// TIA Portal V17 export
// export: Created 2023-09-10T16:27:49.9150522Z, ExportSetting WithDefaults, DisplayName Totally Integrated Automation Portal, DisplayVersion V17, DisplayName TIA Portal Openness, DisplayVersion V17, DisplayName TIA Portal Version Control Interface, DisplayVersion V17, DisplayName STEP 7 Professional, DisplayVersion V17, DisplayName STEP 7 Safety, DisplayVersion V17, DisplayName WinCC Advanced, DisplayVersion V17
ORGANIZATION_BLOCK "Startup"   // OB100, LAD, Startup
TITLE = "Complete Restart"
{ S7_Optimized_Access := 'TRUE' }
VERSION : 0.1
// stored: AutoNumber true, IsIECCheckEnabled false, SetENOAutomatically false
   VAR_INPUT
      LostRetentive : Bool;   // True if retentive data are lost
      LostRTC : Bool;   // True if date and time are lost
   END_VAR
BEGIN

REGION Network 1: modbus Master Init
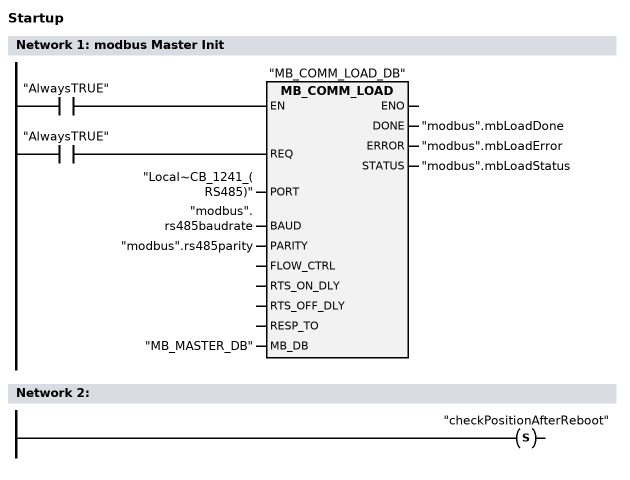
   RUNG wire#powerrail
      Contact( "AlwaysTRUE" )
      "MB_COMM_LOAD_DB".MB_COMM_LOAD(REQ := wire#w1, PORT := "Local~CB_1241_(RS485)", BAUD := "modbus".rs485baudrate, PARITY := "modbus".rs485parity, FLOW_CTRL :=, RTS_ON_DLY :=, RTS_OFF_DLY :=, RESP_TO :=, MB_DB := "MB_MASTER_DB", DONE => "modbus".mbLoadDone, ERROR => "modbus".mbLoadError, STATUS => "modbus".mbLoadStatus)
   END_RUNG
   RUNG wire#powerrail
      Contact( "AlwaysTRUE" )
   END_RUNG wire#w1
   // the same network as SCL:
   IF "AlwaysTRUE" THEN
       "MB_COMM_LOAD_DB"(REQ := "AlwaysTRUE",   // MB_COMM_LOAD
                         PORT := "Local~CB_1241_(RS485)",
                         BAUD := "modbus".rs485baudrate,
                         PARITY := "modbus".rs485parity,
                         MB_DB := "MB_MASTER_DB",
                         DONE => "modbus".mbLoadDone,
                         ERROR => "modbus".mbLoadError,
                         STATUS => "modbus".mbLoadStatus);
   END_IF;
END_REGION

REGION Network 2
   RUNG wire#powerrail
      S_Coil( "checkPositionAfterReboot" )
   END_RUNG
   // the same network as SCL:
   "checkPositionAfterReboot" := TRUE;
END_REGION
END_ORGANIZATION_BLOCK
